FUNCTION F_VolumeToSteps_Path : LREAL
VAR_INPUT
	rVolume    : REAL;       // Requested volume [mL]
    iPumpIndex : UINT;        // Pump index 1..10
    ePath      : E_PumpPath; // Path to apply the correct pump factor
END_VAR
VAR
	rFactor            : REAL;
    rDegreesPerRev     : REAL := 360.0;   // Output expects degrees (1 rev = 360°)
    rEpsilon           : REAL := 1E-6;    // Guard to avoid division by zero
	rRevolutions	   : REAL;
	rRevsPlusHalf	   : REAL;
	iRoundedRevs	   : DINT;
	rFinalDegrees	   : REAL;
END_VAR

// --- Basic input validation ---
IF (iPumpIndex < 1) OR (iPumpIndex > 10) THEN
    // Out of range -> return 0 safely
    F_VolumeToSteps_Path := 0.0;
    RETURN;
END_IF

// --- Select the proper pump factor by path ---
CASE ePath OF
    E_PumpPath.FillJars:
        rFactor := GVL_Motion.aPumps[iPumpIndex].Rotary.rPumpFactorFillJars;
    E_PumpPath.FillCalBox:
        rFactor := GVL_Motion.aPumps[iPumpIndex].Rotary.rPumpFactorFillCalBox;
    E_PumpPath.FromCalBox:
        rFactor := GVL_Motion.aPumps[iPumpIndex].Rotary.rPumpFactorFromCalBox;
ELSE
    // Fallback (defensive): default to FillJars
    rFactor := GVL_Motion.aPumps[iPumpIndex].Rotary.rPumpFactorFillJars;
END_CASE

// --- Guard against invalid/zero factor ---
IF ABS(rFactor) <= rEpsilon THEN
    // Factor not calibrated -> return 0 safely
    F_VolumeToSteps_Path := 0.0;
    RETURN;
END_IF

// 1. Calculate the required number of revolutions (pode ser fracionário)
// Revolutions = Volume [mL] / Factor [mL/rev]
rRevolutions := rVolume / rFactor;

// 2. Implement the rounding logic: TRUNC(x + 0.5)
rRevsPlusHalf := rRevolutions + 0.5;

// 3. Truncate the value to get the nearest integer revolution count.
iRoundedRevs := REAL_TO_DINT(TRUNC(rRevsPlusHalf));

// 4. Convert the integer revolutions back to the angular distance in degrees.
rFinalDegrees := DINT_TO_REAL(iRoundedRevs) * rDegreesPerRev;

// --- Return the final angular distance (in degrees) as LREAL for motion control ---
F_VolumeToSteps_Path := REAL_TO_LREAL(rFinalDegrees);

END_FUNCTION

(* stored: Version 1.1.0.1, ProductVersion 3.1.4024.15
   POU F_VolumeToSteps_Path: Id {c202cb0f-adf8-4c38-b92d-fd44fa4ca689}, SpecialFunc None *)
